// TwinCAT 3 PLC project Untitled1
// ProgramVersion: 3.1.4023.0
// libraries:
//   Tc2_Standard, * (Beckhoff Automation GmbH)
//   Tc2_System, * (Beckhoff Automation GmbH)
//   Tc3_EventLogger, * (Beckhoff Automation GmbH)
//   Tc3_Module, * (Beckhoff Automation GmbH)
// project tree:
//   DUTs/ E_Operator.TcDUT, Parameter.TcDUT, ST_MyStruct.TcDUT
//   GVLs/ GVL.TcGVL, Parameters.TcGVL
//   / PlcTask.TcTTO
//   POUs/ FB_Base.TcPOU, FB_ExtBase.TcPOU, MAIN.TcPOU, MAIN_1.TcPOU
// real-time tasks:
//   TASK PlcTask: cycle T#10ms, priority 20, ADS port 350

CONFIGURATION Untitled1
    RESOURCE PLC ON TwinCAT3
        TASK PlcTask(INTERVAL := T#10ms, PRIORITY := 20);
        PROGRAM MAIN WITH PlcTask : MAIN;
    END_RESOURCE
END_CONFIGURATION

// ---- DUTs/E_Operator.TcDUT
{attribute 'qualified_only'}
{attribute 'strict'}
TYPE E_Operator :
(
	idle_operator := 0,
	sum_operator,
	diff_operator,
	mul_operator,
	ratio_operator
);
END_TYPE

// ---- DUTs/Parameter.TcDUT
TYPE Parameter :
STRUCT
	Value : REAL;				//Value to input
	StoredValue : REAL;			//Value to store data if it is valid
	Minimun, Maximun : REAL;	//Min/Max valid range
	nDecpt : INT;				//Number of decimal digit
	Description : STRING;		//Parameter description
END_STRUCT
END_TYPE

// ---- DUTs/ST_MyStruct.TcDUT
TYPE ST_MyStruct :
STRUCT
	A, B, C : INT;
	Value : REAL;
	Descr : STRING;
END_STRUCT
END_TYPE

// ---- GVLs/GVL.TcGVL
{attribute 'qualified_only'}
VAR_GLOBAL
	arrStruct : ARRAY [0..9] OF ST_MyStruct;
	arrReal : ARRAY [0..9] OF REAL;
	iTest : INT;
	rTest : REAL;
END_VAR

// ---- GVLs/Parameters.TcGVL
{attribute 'qualified_only'}
VAR_GLOBAL
	//Lista of single structure variables
	rParameter01 : Parameter;
	rParameter02 : Parameter;
	rParameter03 : Parameter;
	rParameter04 : Parameter;
	rParameter05 : Parameter;
	rParameter06 : Parameter;
	rParameter07 : Parameter;
	rParameter08 : Parameter;
	
	//Array of structures
	aParameters : ARRAY [0..9] OF Parameter;
END_VAR

// ---- POUs/MAIN.TcPOU
PROGRAM MAIN
VAR
	bInit: BOOL;
	i: INT;
	j: INT;
	
	// FB Instances
	Base : FB_Base;			//Base FB
	ExtBase : FB_ExtBase;	//Extended FB	
END_VAR

IF bInit = FALSE THEN
	bInit := TRUE;
	Parameters.rParameter01.Description := 'parametro 1';
	Parameters.rParameter01.Maximun := 1000;
	Parameters.rParameter01.Minimun := -1000;
	Parameters.rParameter01.nDecpt := 2;
	
	Parameters.rParameter02.Description := 'parametro 2';
	Parameters.rParameter02.Maximun := 1000;
	Parameters.rParameter02.Minimun := 0;
	Parameters.rParameter02.nDecpt := 2;
	
	Parameters.rParameter03.Description := 'parametro 3';
	Parameters.rParameter03.Maximun := 1000;
	Parameters.rParameter03.Minimun := -1000;
	Parameters.rParameter03.nDecpt := 2;
	
	Parameters.rParameter04.Description := 'parametro 4';
	Parameters.rParameter04.Maximun := 10;
	Parameters.rParameter04.Minimun := -5;
	Parameters.rParameter04.nDecpt := 2;
	
	Parameters.rParameter05.Description := 'parametro 5';
	Parameters.rParameter05.Maximun := 1000;
	Parameters.rParameter05.Minimun := -1000;
	Parameters.rParameter05.nDecpt := 4;
	
	Parameters.rParameter06.Description := 'parametro 6';
	Parameters.rParameter06.Maximun := 123;
	Parameters.rParameter06.Minimun := -1;
	Parameters.rParameter06.nDecpt := 2;
	
	Parameters.rParameter07.Description := 'parametro 7';
	Parameters.rParameter07.Maximun := 1000;
	Parameters.rParameter07.Minimun := -1000;
	Parameters.rParameter07.nDecpt := 3;
	
	Parameters.rParameter08.Description := 'parametro 8';
	Parameters.rParameter08.Maximun := 1000;
	Parameters.rParameter08.Minimun := -1000;
	Parameters.rParameter08.nDecpt := 2;
	FOR i := 0 TO 9 DO
		GVL.arrReal[i] := i;
		GVL.arrStruct[i].A := i;
		GVL.arrStruct[i].B := i;
		GVL.arrStruct[i].C := i;
		GVL.arrStruct[i].Value := i;
		GVL.arrStruct[i].Descr := INT_TO_STRING(i);
		
		Parameters.aParameters[i].Description := Concat('Parametro', INT_TO_STRING(i));
		Parameters.aParameters[i].Value := i;
		Parameters.aParameters[i].StoredValue := i;
		Parameters.aParameters[i].Maximun := 1000;
		Parameters.aParameters[i].Minimun := -10;
	END_FOR	
END_IF

MAIN_1();

END_PROGRAM

// ---- POUs/FB_Base.TcPOU
FUNCTION_BLOCK FB_Base
VAR_INPUT
END_VAR
VAR_OUTPUT
END_VAR
VAR
	_CalcCounter : INT;
END_VAR

{attribute 'monitoring' := 'call'}
PROPERTY CalcCounter : INT
GET
CalcCounter := _CalcCounter;
END_GET
SET
_CalcCounter := CalcCounter;
END_SET
END_PROPERTY

{attribute 'TcRpcEnable'}
METHOD Calculation : REAL
VAR_INPUT	
	in1, in2 : REAL;
	operator : E_Operator;
END_VAR
CASE operator OF
	E_Operator.idle_operator:
		;
	E_Operator.sum_operator:
		Calculation := in1 + in2;
	E_Operator.diff_operator:
		Calculation := in1 - in2;
	E_Operator.mul_operator:
		Calculation := in1 * in2;
	E_Operator.ratio_operator:
		IF in2 <> 0 THEN
			Calculation := in1 / in2;
		END_IF	
END_CASE
_CalcCounter := _CalcCounter + 1;
END_METHOD

END_FUNCTION_BLOCK

// ---- POUs/FB_ExtBase.TcPOU
FUNCTION_BLOCK FB_ExtBase EXTENDS FB_Base
VAR_INPUT
END_VAR
VAR_OUTPUT
END_VAR
VAR
END_VAR

{attribute 'monitoring' := 'call'}
PROPERTY CalcCounter : INT
GET
END_GET
END_PROPERTY

{attribute 'TcRpcEnable'}
METHOD ResetCalcCounter : BOOL
VAR_INPUT
END_VAR
_CalcCounter := 0;
END_METHOD

END_FUNCTION_BLOCK

// ---- POUs/MAIN_1.TcPOU
PROGRAM MAIN_1
VAR
	fbEventlogger : FB_TcEventLogger;
	fbAlarm: FB_TcAlarm;
	fbMessage: FB_TcMessage;
	
	bAlarm: BOOL;
	bMessage : BOOL;
	bIsInitalized: BOOL;
	bClearAlarm: BOOL;
	bConfirmAlarm: BOOL;
END_VAR

IF NOT bIsInitalized THEN
	bIsInitalized := TRUE;
	fbMessage.CreateEx(TC_Events.MyEvents.Start, 0);
	fbAlarm.CreateEx(TC_Events.MyEvents.Stop, TRUE, 0);
END_IF

IF bMessage THEN
	bMessage := FALSE;
	fbMessage.Send(0);
END_IF

IF bAlarm THEN
	bAlarm := FALSE;
	fbAlarm.Raise(0);
END_IF

IF bClearAlarm THEN
	bClearAlarm := FALSE;
	fbAlarm.Clear(0, TRUE);
END_IF

END_PROGRAM
